(* PLC project Blank Project, Blank Blank 1.0 *)
(* stored: creationDateTime 2016-05-18T21:14:07, modificationDateTime 2016-12-15T19:37:15 *)

PROGRAM My_Program
  VAR
    transformer AT %QX0.0 : BOOL := 1;
    switch1 AT %QW0 : INT := 0;
    switch2 AT %QW1 : INT := 1;
    switch3 AT %QW2 : INT := 0;
  END_VAR

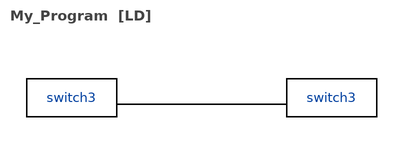
(* LD diagram, written out as Structured Text *)
switch3 := switch3;
END_PROGRAM

CONFIGURATION Config0
  RESOURCE Res0 ON PLC
    TASK TaskMain(INTERVAL := T#50ms, PRIORITY := 0);
    PROGRAM Inst0 WITH TaskMain : My_Program;
  END_RESOURCE
END_CONFIGURATION
